FUNCTION "JsonW_LNK_Fixture" : Void
{ S7_Optimized_Access := 'TRUE' }
VERSION : 0.1
   VAR_IN_OUT
      Buf : Array[*] of Byte;   // 출력 버퍼
      Pos : DInt;   // 다음 쓸 절대 인덱스 (< 0 = 오류 유지)
      Val : "LNK_Fixture";   // 쓸 값
   END_VAR

   VAR_TEMP
      i0 : DInt;
      i1 : DInt;
   END_VAR


BEGIN
	// GENERATED by gr-contract gen-link from "LNK_Fixture" sig 16#EB2E5DE0 - do not edit
	// wire-spec 2 : 선언 순서, 공백 없음. 버퍼가 모자라면 Pos := LNK_JERR_OVERFLOW (끈끈한 오류, 호출자가 끝에 한 번 확인)
	"Json_WRaw"(Buf := #Buf, Pos := #Pos, Lit := '{"B0":');
	"Json_WBool"(Buf := #Buf, Pos := #Pos, Val := #Val.B0);
	"Json_WRaw"(Buf := #Buf, Pos := #Pos, Lit := ',"B1":');
	"Json_WBool"(Buf := #Buf, Pos := #Pos, Val := #Val.B1);
	"Json_WRaw"(Buf := #Buf, Pos := #Pos, Lit := ',"B2":');
	"Json_WBool"(Buf := #Buf, Pos := #Pos, Val := #Val.B2);
	"Json_WRaw"(Buf := #Buf, Pos := #Pos, Lit := ',"B3":');
	"Json_WBool"(Buf := #Buf, Pos := #Pos, Val := #Val.B3);
	"Json_WRaw"(Buf := #Buf, Pos := #Pos, Lit := ',"B4":');
	"Json_WBool"(Buf := #Buf, Pos := #Pos, Val := #Val.B4);
	"Json_WRaw"(Buf := #Buf, Pos := #Pos, Lit := ',"B5":');
	"Json_WBool"(Buf := #Buf, Pos := #Pos, Val := #Val.B5);
	"Json_WRaw"(Buf := #Buf, Pos := #Pos, Lit := ',"B6":');
	"Json_WBool"(Buf := #Buf, Pos := #Pos, Val := #Val.B6);
	"Json_WRaw"(Buf := #Buf, Pos := #Pos, Lit := ',"B7":');
	"Json_WBool"(Buf := #Buf, Pos := #Pos, Val := #Val.B7);
	"Json_WRaw"(Buf := #Buf, Pos := #Pos, Lit := ',"B8":');
	"Json_WBool"(Buf := #Buf, Pos := #Pos, Val := #Val.B8);
	"Json_WRaw"(Buf := #Buf, Pos := #Pos, Lit := ',"By":');
	"Json_WByte"(Buf := #Buf, Pos := #Pos, Val := #Val."By");
	"Json_WRaw"(Buf := #Buf, Pos := #Pos, Lit := ',"Si":');
	"Json_WSInt"(Buf := #Buf, Pos := #Pos, Val := #Val.Si);
	"Json_WRaw"(Buf := #Buf, Pos := #Pos, Lit := ',"I":');
	"Json_WInt"(Buf := #Buf, Pos := #Pos, Val := #Val.I);
	"Json_WRaw"(Buf := #Buf, Pos := #Pos, Lit := ',"W":');
	"Json_WWord"(Buf := #Buf, Pos := #Pos, Val := #Val.W);
	"Json_WRaw"(Buf := #Buf, Pos := #Pos, Lit := ',"Di":');
	"Json_WDInt"(Buf := #Buf, Pos := #Pos, Val := #Val.Di);
	"Json_WRaw"(Buf := #Buf, Pos := #Pos, Lit := ',"Udi":');
	"Json_WUDInt"(Buf := #Buf, Pos := #Pos, Val := #Val.Udi);
	"Json_WRaw"(Buf := #Buf, Pos := #Pos, Lit := ',"R":');
	"Json_WReal"(Buf := #Buf, Pos := #Pos, Val := #Val.R);
	"Json_WRaw"(Buf := #Buf, Pos := #Pos, Lit := ',"Lr":');
	"Json_WLReal"(Buf := #Buf, Pos := #Pos, Val := #Val.Lr);
	"Json_WRaw"(Buf := #Buf, Pos := #Pos, Lit := ',"Li":');
	"Json_WLInt"(Buf := #Buf, Pos := #Pos, Val := #Val.Li);
	"Json_WRaw"(Buf := #Buf, Pos := #Pos, Lit := ',"Ch":');
	"Json_WChar"(Buf := #Buf, Pos := #Pos, Val := #Val.Ch);
	"Json_WRaw"(Buf := #Buf, Pos := #Pos, Lit := ',"Str":');
	"Json_WStr"(Buf := #Buf, Pos := #Pos, Val := #Val.Str);
	"Json_WRaw"(Buf := #Buf, Pos := #Pos, Lit := ',"Ts":');
	"Json_WDtl"(Buf := #Buf, Pos := #Pos, Val := #Val.Ts);
	"Json_WRaw"(Buf := #Buf, Pos := #Pos, Lit := ',"Tm":');
	"Json_WTime"(Buf := #Buf, Pos := #Pos, Val := #Val.Tm);
	"Json_WRaw"(Buf := #Buf, Pos := #Pos, Lit := ',"Flags":[');
	FOR #i0 := 0 TO 2 DO
	  IF #i0 > 0 THEN
	    "Json_WComma"(Buf := #Buf, Pos := #Pos);
	  END_IF;
	  "Json_WBool"(Buf := #Buf, Pos := #Pos, Val := #Val.Flags[#i0]);
	END_FOR;
	"Json_WRaw"(Buf := #Buf, Pos := #Pos, Lit := '],"Axis":[');
	FOR #i0 := 1 TO 3 DO   // "X".."Z"
	  IF #i0 > 1 THEN
	    "Json_WComma"(Buf := #Buf, Pos := #Pos);
	  END_IF;
	  "Json_WReal"(Buf := #Buf, Pos := #Pos, Val := #Val.Axis[#i0]);
	END_FOR;
	"Json_WRaw"(Buf := #Buf, Pos := #Pos, Lit := '],"Grid":[');
	FOR #i0 := 1 TO 2 DO
	  IF #i0 > 1 THEN
	    "Json_WRaw"(Buf := #Buf, Pos := #Pos, Lit := ',[');
	  ELSE
	    "Json_WRaw"(Buf := #Buf, Pos := #Pos, Lit := '[');
	  END_IF;
	  FOR #i1 := 0 TO 1 DO
	    IF #i1 > 0 THEN
	      "Json_WComma"(Buf := #Buf, Pos := #Pos);
	    END_IF;
	    "Json_WInt"(Buf := #Buf, Pos := #Pos, Val := #Val.Grid[#i0, #i1]);
	  END_FOR;
	  "Json_WRaw"(Buf := #Buf, Pos := #Pos, Lit := ']');
	END_FOR;
	"Json_WRaw"(Buf := #Buf, Pos := #Pos, Lit := '],"Outer":{"A":');
	"Json_WUSInt"(Buf := #Buf, Pos := #Pos, Val := #Val.Outer.A);
	"Json_WRaw"(Buf := #Buf, Pos := #Pos, Lit := ',"Inner":{"Flag":');
	"Json_WBool"(Buf := #Buf, Pos := #Pos, Val := #Val.Outer.Inner.Flag);
	"Json_WRaw"(Buf := #Buf, Pos := #Pos, Lit := ',"Val":');
	"Json_WUInt"(Buf := #Buf, Pos := #Pos, Val := #Val.Outer.Inner.Val);
	"Json_WRaw"(Buf := #Buf, Pos := #Pos, Lit := '}},"Sub":');
	"JsonW_LNK_FixtureSub"(Buf := #Buf, Pos := #Pos, Val := #Val.Sub);
	"Json_WRaw"(Buf := #Buf, Pos := #Pos, Lit := ',"Subs":[');
	FOR #i0 := 0 TO 1 DO
	  IF #i0 > 0 THEN
	    "Json_WComma"(Buf := #Buf, Pos := #Pos);
	  END_IF;
	  "JsonW_LNK_FixtureSub"(Buf := #Buf, Pos := #Pos, Val := #Val.Subs[#i0]);
	END_FOR;
	"Json_WRaw"(Buf := #Buf, Pos := #Pos, Lit := ']}');
END_FUNCTION
